VAR_GLOBAL
    KommAnVisu                 : INT;      (* Kommunikation an die Visualisierung *)
    KommVonVisu                : INT;      (* Kommunikation von der Visualisierung *)
    belegt                     : BOOL;     (* true = erzeugt Dummyteil, false = keine Auswirkungen (nur Handauflage) *)
    daten_gebucht              : BOOL;
    SteuerStatus               : DUT_Visu_SteuerStatus;

    // Frequenzumrichter
	Trans_Schlossseite			: DUT_SEW_FU_Visu; 		//#Tab: 3510 Transport #Name: Transport Schlossseite X-Achse

    // Servoregler
	X_Achse						: DUT_Achse_Service;	//#Tab: 3510 Transport #Name: X-Achse Längsanschlag

    // Ventile
	 Laengsanschl        		: DUT_Ventil_VISU;      //#Tab: 3510 Transport #Name: Schlossseite Längsanschlag
	 Schienenklemm        		: DUT_Ventil_VISU;      //#Tab: 3510 Transport #Name: Schienenklemmung

END_VAR

VAR_GLOBAL PERSISTENT
    Schrittnummer           : INT;
    Kopfdaten               : DUT_Kopfdaten;
    Kopfdaten_default       : DUT_Kopfdaten;
    Jobdaten                : ARRAY[1..10] OF DUT_Jobdaten;
    Jobdaten_default        : ARRAY[1..10] OF DUT_Jobdaten;
	aktJob					: DUT_Jobdaten;

    //para_Vorlage             : REAL := 0.0; //#Typ: VParam #Tab:  #Name:  #Einheit:mm #Min: 1 #Max: 100 #Format:F1
END_VAR

(* stored: Version 1.1.0.1
   GVL GVL_Visu_3510: Id {4fbf8656-4b4c-4d82-a6c7-93df2eeee22a} *)
